PROGRAM BackgroundRS422
VAR
END_VAR

BackgroundEL6021();

END_PROGRAM

(* stored: Version 1.1.0.1, ProductVersion 3.1.4024.12
   POU BackgroundRS422: Id {93f68232-d285-4c23-bd55-21756aa79839}, SpecialFunc None *)
